PROGRAM MainControl
VAR
	fbErrorHandling : FB_ErrorHandling;
	fbServiceModule : FB_ServiceModule;
	fbLevitationSystem : FB_LevitationSystem;
	fbGuidanceSystem : FB_GuidanceSystem;
	


	
	eMainState : eMainStateMachine := eMainStateMachine.STARTUP;
	fbErrorTimer : TON;										//10s
	stMode : stOperationMode;
END_VAR


CASE eMainState OF
	
	eMainStateMachine.STARTUP:
	
		IF stMode.eMode = eOperationMode.RUN THEN
			doCheckSystem();
		ELSIF stMode.eMode = eOperationMode.TEST THEN
			stMode.nTestMode.0 := stMode.bTestServiceModule;
			stMode.nTestMode.1 := stMode.bTestLevitationSystem;
			stMode.nTestMode.2 := stMode.bTestGuidanceSystem;
			
			CASE stMode.nTestMode OF
				0:
					fbServiceModule.setSLEEP := TRUE;
					fbLevitationSystem.setSLEEP := TRUE;
					fbGuidanceSystem.setSLEEP := TRUE;
				1:
					fbServiceModule.setSLEEP := FALSE;
					fbLevitationSystem.setSLEEP := TRUE;
					fbGuidanceSystem.setSLEEP := TRUE;
				2:
					fbServiceModule.setSLEEP := TRUE;
					fbLevitationSystem.setSLEEP := FALSE;
					fbGuidanceSystem.setSLEEP := TRUE;
				3:
					fbServiceModule.setSLEEP := FALSE;
					fbLevitationSystem.setSLEEP := FALSE;
					fbGuidanceSystem.setSLEEP := TRUE;
				4:
					fbServiceModule.setSLEEP := TRUE;
					fbLevitationSystem.setSLEEP := TRUE;
					fbGuidanceSystem.setSLEEP := FALSE;
				5:
					fbServiceModule.setSLEEP := FALSE;
					fbLevitationSystem.setSLEEP := TRUE;
					fbGuidanceSystem.setSLEEP := FALSE;
				6:
					fbServiceModule.setSLEEP := TRUE;
					fbLevitationSystem.setSLEEP := FALSE;
					fbGuidanceSystem.setSLEEP := FALSE;
				7:
					fbServiceModule.setSLEEP := FALSE;
					fbLevitationSystem.setSLEEP := FALSE;
					fbGuidanceSystem.setSLEEP := FALSE;
			END_CASE
			
			doCheckSystem();
		END_IF
		
		
	eMainStateMachine.READY:
		iTest := 2;

	eMainStateMachine.OPERATIONAL:
		iTest := 3;

	eMainStatemachine.SHUTDOWN:
		iTest := 4;

	eMainStateMachine.ERROR:
		iTest := 5;	




END_CASE

METHOD doCheckSystem
VAR_INPUT
END_VAR
VAR
END_VAR
fbErrorHandling();
fbServiceModule();
fbLevitationSystem();
fbGuidanceSystem();
		
IF (fbServiceModule.eCondition = eConditionCheck.READY OR fbServiceModule.eCondition = eConditionCheck.SLEEP) AND (fbLevitationSystem.eCondition = eConditionCheck.READY OR fbLevitationSystem.eCondition = eConditionCheck.SLEEP) AND (fbGuidanceSystem.eCondition = eConditionCheck.READY OR fbGuidanceSystem.eCondition = eConditionCheck.SLEEP) THEN
	eMainState := eMainStateMachine.READY;
ELSIF fbServiceModule.eCondition = eConditionCheck.ERROR OR fbLevitationSystem.eCondition = eConditionCheck.ERROR OR fbGuidanceSystem.eCondition = eConditionCheck.ERROR THEN
	fbErrorTimer(IN := TRUE, PT := T#10S);
	IF fbErrorTimer.Q THEN
		fbErrorTimer.IN := FALSE;
		eMainState := eMainStateMachine.ERROR;
	END_IF
ELSE
	fbErrorTimer.IN := FALSE;
	eMainState := eMainStateMachine.STARTUP;
END_IF
END_METHOD

END_PROGRAM

(* stored: Version 1.1.0.1, ProductVersion 3.1.4024.12
   POU MainControl: Id {165fa4b6-fe79-4748-9022-b33b5b722466}, SpecialFunc None
   Method doCheckSystem: Id {55b5a3ff-6d8a-4578-a9a0-1bbfe6d7f606} *)
